// Mitsubishi GX Developer project: Станок производства уголка   PLC: FX3G

PROGRAM MAIN
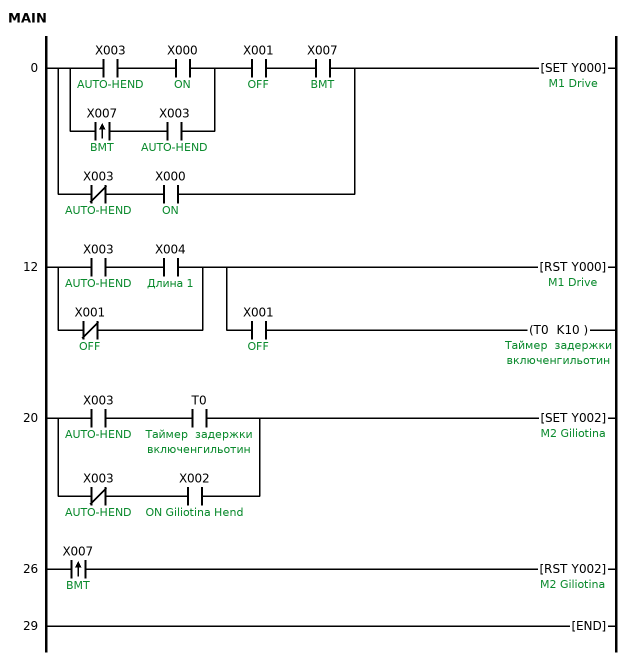
0     LD      X003  ; AUTO-HEND
      AND     X000  ; ON
      LDP     X007  ; ВМТ
      AND     X003  ; AUTO-HEND
      ORB
      AND     X001  ; OFF
      AND     X007  ; ВМТ
      LDI     X003  ; AUTO-HEND
      AND     X000  ; ON
      ORB
      SET     Y000  ; M1 Drive
12    LD      X003  ; AUTO-HEND
      AND     X004  ; Длина 1
      ORI     X001  ; OFF
      RST     Y000  ; M1 Drive
      AND     X001  ; OFF
      OUT     T0 K10  ; Таймер  задержки включенгильотин
20    LD      X003  ; AUTO-HEND
      AND     T0  ; Таймер  задержки включенгильотин
      LDI     X003  ; AUTO-HEND
      AND     X002  ; ON Giliotina Hend
      ORB
      SET     Y002  ; M2 Giliotina
26    LDP     X007  ; ВМТ
      RST     Y002  ; M2 Giliotina
29    END
END_PROGRAM

// device comments not shown above
X005  ; Длина 2
X006  ; Длина 3
Y001  ; M1 Drive Jog
